{attribute 'qualified_only'}
{attribute 'strict'}
TYPE Bumperstatus :
(
	init,
	normal,
	triggered
);
END_TYPE

(* stored: Version 1.1.0.1, ProductVersion 3.1.4024.11
   DUT Bumperstatus: Id {954f804d-f325-4abb-afde-f79ab9cf891f} *)
